PROGRAM MAIN
VAR
END_VAR

A_Program();
B_Program();

END_PROGRAM

(* stored: Version 1.1.0.1, ProductVersion 3.1.4025.12
   POU MAIN: Id {db0ea7e8-4270-46be-a1fa-23f9fadb01ec}, SpecialFunc None *)
